FUNCTION_BLOCK ServoHandling
VAR_INPUT
END_VAR
VAR_OUTPUT
END_VAR
VAR
  	// Alarm inputs from Axis
  	XAxisAlarm AT %I*:BOOL := TRUE;
  	YAxisAlarm AT %I*:BOOL := TRUE;
  	ZAxisAlarm AT %I*:BOOL := TRUE;
  	AAxisAlarm AT %I*:BOOL := TRUE;
  	// Alarm Output to PC pin 8
  	PCServoAlarm AT %Q*:BOOL := FALSE;
	
  	// Whether servo thinks Z Axis break should be off
  	ZAxisBrakeOff AT %I*:BOOL := FALSE;
	// Relay output controlling ZAxis Brake
	ZAxisBrakeRelay AT %Q*: BOOL := FALSE;
END_VAR

PCServoAlarm := XAxisAlarm AND YAxisAlarm AND ZAxisAlarm AND AAxisAlarm;
ZAxisBrakeRelay := ZAxisBrakeOff;

END_FUNCTION_BLOCK

(* stored: Version 1.1.0.1, ProductVersion 3.1.4022.12
   POU ServoHandling: Id {8a13316b-cf16-4b49-a13c-85ac385b3e37}, SpecialFunc None *)
